TEXTLIST TextList_Przyciski_Menu
  0 = 'GŁÓWNA'
  1 = 'ALARMY'
  2 = 'USTAWIENIA'
   = ''
END_TEXTLIST

(* stored: Version 1.1.0.1, ProductVersion 3.1.4024.15
   TextList TextList_Przyciski_Menu: Id {973f32f2-3b49-419f-a10c-b29903459bde} *)
